FUNCTION TEST_FINISHED : BOOL
VAR
    TestName : Tc2_System.T_MaxString;
    Counter : UINT := 0;
END_VAR

// Grab the currently running test name
TestName := GVL_TcUnit.CurrentTestNameBeingCalled;

TEST_FINISHED := FALSE;
// Find the test suite and set the test as finished
FOR Counter := 1 TO GVL_TcUnit.NumberOfInitializedTestSuites BY 1 DO
    IF GVL_TcUnit.TestSuiteAddresses[Counter] = GVL_TcUnit.CurrentTestSuiteBeingCalled THEN
        GVL_TcUnit.TestSuiteAddresses[Counter]^.SetTestFinished(TestName := GVL_TcUnit.CurrentTestNameBeingCalled);
        TEST_FINISHED := TRUE;
        RETURN;
    END_IF
END_FOR

END_FUNCTION

(* stored: Version 1.1.0.1, ProductVersion 3.1.4022.18
   POU TEST_FINISHED: Id {9922b45b-fca5-4323-be8f-93710371a816}, SpecialFunc None *)
